{attribute 'GeneratedUsingTerminal: EL5072-0000-0016'}
{attribute addProperty BoxType "EL5072-0000-0016"}
{attribute addProperty Id "StatusAT %I*Status_3673109410PositionAT %I*DINT4Latch_valueAT %I*DINT4"}
{attribute addProperty CRC "3152560159"}
{attribute addProperty Size "18"}
TYPE IND_Inputs_Channel_BBE8401F EXTENDS InputBase_8311D824 :
STRUCT
	{attribute addProperty Name "Status"}
	Status AT %I* : Status_36731094;
	{attribute addProperty Name "Position"}
	Position AT %I* : DINT;
	{attribute addProperty Name "Latch_value"}
	Latch_value AT %I* : DINT;
END_STRUCT
END_TYPE

(* stored: Version 1.2.0.0, ProductVersion 3.1.4024.11
   DUT IND_Inputs_Channel_BBE8401F: Id {3a85af14-ea09-4dbe-b42d-5f227673c07a} *)
